SUBAPPLICATION Uebung_172b_ASRT (* Exercise for ASRT_AX_T_FF_SR, ueber AE-Adapter statt rohe Events (ASRT_3AE_TO_SRT statt ASRT_3EVENTS_TO_SRT) *)
  (* Standard: 61499-2; Description: Copyright (c) 2026 Meisterschulen am Ostbahnhof This program and the accompanying materials are made available under the terms of the Eclipse Public License 2.0 which is available at https://www.eclipse.org/legal/epl-2.0/ SPDX-License-Identifier: EPL-2.0 *)
  (* Version 1.0, 2026-09-07, Franz Höpfinger, Meisterschulen am Ostbahnhof, initial API and implementation and/or initial documentation *)
  PACKAGE Uebungen;
  IMPORT logiBUS::io::DI::logiBUS_DI::Input_I1;
  IMPORT logiBUS::io::DI::logiBUS_DI::Input_I2;
  IMPORT logiBUS::io::DI::logiBUS_DI::Input_I3;
  IMPORT logiBUS::io::DI::logiBUS_DI_Events::BUTTON_SINGLE_CLICK;
  IMPORT logiBUS::io::DQ::logiBUS_DO::Output_Q1;
  (* Documentation:
  SET/RESET/TOGGLE über AE-Adapter statt rohe Events
   Dieselbe Funktion wie Uebung_172_ASRT (I1 = SET-Klick, I2 = RESET-Klick, I3 = TOGGLE-Klick, Latch via ASRT_AX_T_FF_SR), aber der Umweg über ASRT_3AE_TO_SRT statt ASRT_3EVENTS_TO_SRT zeigt, WARUM es den AE-Adapter-Weg überhaupt gibt.
   Funktionsbeschreibung
    - ASRT_3EVENTS_TO_SRT (in Uebung_172_ASRT) hat rohe EventInputs - jede beliebige Event-Quelle passt direkt, ohne Typ-Zwang, aber auch ohne dass sich das Signal wie ein Adapter weiterverarbeiten lässt.
   - ASRT_3AE_TO_SRT hat stattdessen SET_IN/RESET_IN/ TOGGLE_IN als AE-Adapter-Sockets - jede Quelle muss selbst einen AE-Plug liefern. Je ein AE_EVENT_TO_E baut die Brücke: rohes Klick-Event (logiBUS_IE.IND) hinein, getypter AE-Plug heraus.
   - Der Gewinn: ein AE-Plug ist ein normaler Adapter wie AX/ASR/ASRT - er lässt sich mit AE_SPLIT_2 vervielfältigen oder zusammenführen, genau wie es Uebung_231_AX für ASR zeigt. Ein rohes Event kann das nicht.
    Arbeitsauftrag
   Testen Sie identisch zu Uebung_172_ASRT: I1 klicken → Q1 EIN, I2 klicken → Q1 AUS, I3 klicken → Q1 wechselt den Zustand. Vergleichen Sie im Editor beide SubApps - gleiches Verhalten, aber Uebung_172b_ASRT hat zwischen Tastern und Latch drei zusätzliche AE_EVENT_TO_E-Bausteine.
  *)
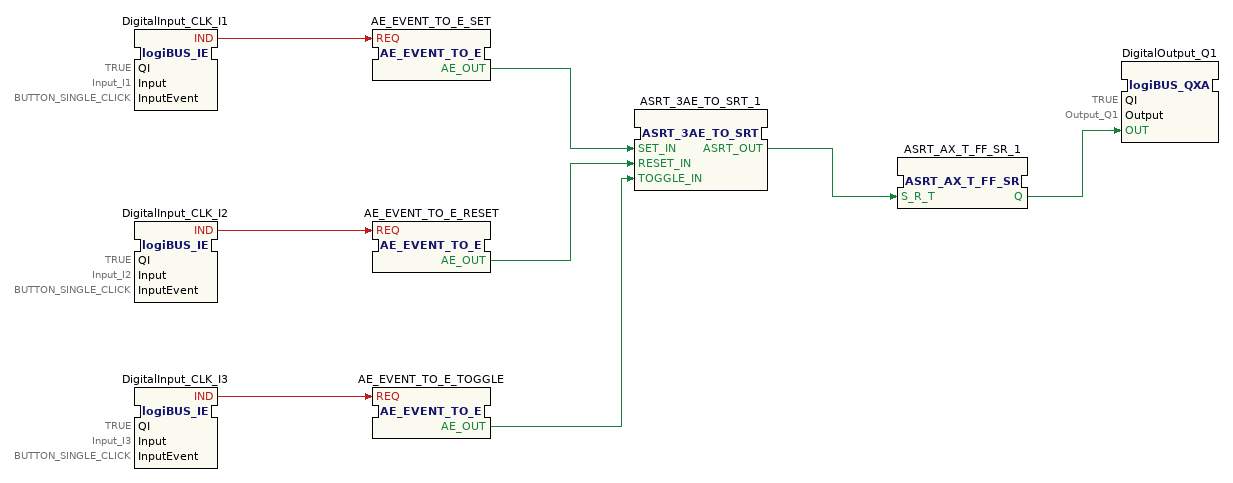
  (* Vergleich zu Uebung_172_ASRT: dort ASRT_3EVENTS_TO_SRT mit rohen EventInputs (jede beliebige Quelle passt, ohne Typ). Hier ASRT_3AE_TO_SRT mit AE-Adapter-Sockets: jede Quelle muss selbst einen AE-Plug liefern - AE_EVENT_TO_E baut je Kanal die Bruecke vom rohen Klick-Event zum typisierten AE. Vorteil: AE-Plugs lassen sich wie jeder Adapter mit AE_SPLIT_2 vervielfaeltigen oder zusammenfuehren, ein rohes Event nicht. *)
  FBS
    ASRT_AX_T_FF_SR_1 : adapter::events::unidirectional::ASRT_AX_T_FF_SR;
    ASRT_3AE_TO_SRT_1 : adapter::conversion::unidirectional::ASRT_3AE_TO_SRT;
    AE_EVENT_TO_E_SET : adapter::conversion::unidirectional::AE_EVENT_TO_E;
    AE_EVENT_TO_E_RESET : adapter::conversion::unidirectional::AE_EVENT_TO_E;
    AE_EVENT_TO_E_TOGGLE : adapter::conversion::unidirectional::AE_EVENT_TO_E;
    DigitalInput_CLK_I1 : logiBUS::io::DI::logiBUS_IE(QI := TRUE, Input := Input_I1, InputEvent := BUTTON_SINGLE_CLICK);
    DigitalOutput_Q1 : logiBUS::io::DQ::logiBUS_QXA(QI := TRUE, Output := Output_Q1);
    DigitalInput_CLK_I2 : logiBUS::io::DI::logiBUS_IE(QI := TRUE, Input := Input_I2, InputEvent := BUTTON_SINGLE_CLICK);
    DigitalInput_CLK_I3 : logiBUS::io::DI::logiBUS_IE(QI := TRUE, Input := Input_I3, InputEvent := BUTTON_SINGLE_CLICK);
  END_FBS
  EVENT_CONNECTIONS
    DigitalInput_CLK_I1.IND TO AE_EVENT_TO_E_SET.REQ;
    DigitalInput_CLK_I2.IND TO AE_EVENT_TO_E_RESET.REQ;
    DigitalInput_CLK_I3.IND TO AE_EVENT_TO_E_TOGGLE.REQ;
  END_CONNECTIONS
  ADAPTER_CONNECTIONS
    AE_EVENT_TO_E_SET.AE_OUT TO ASRT_3AE_TO_SRT_1.SET_IN;
    AE_EVENT_TO_E_RESET.AE_OUT TO ASRT_3AE_TO_SRT_1.RESET_IN;
    AE_EVENT_TO_E_TOGGLE.AE_OUT TO ASRT_3AE_TO_SRT_1.TOGGLE_IN;
    ASRT_3AE_TO_SRT_1.ASRT_OUT TO ASRT_AX_T_FF_SR_1.S_R_T;
    ASRT_AX_T_FF_SR_1.Q TO DigitalOutput_Q1.OUT;
  END_CONNECTIONS
END_SUBAPPLICATION
